INTERFACE I_EventHandler

METHOD PUBLIC HandleEvent
VAR_INPUT
	Event : I_Event;
END_VAR
END_METHOD

END_INTERFACE

(* stored: Version 1.1.0.1, ProductVersion 3.1.4024.12
   Itf I_EventHandler: Id {c10c7a89-e538-0400-2961-b798e996977b}
   Method HandleEvent: Id {4fb476c4-d3ce-0d9a-0666-a1a8dfc174ac} *)
